(* PLC project FBDexample, Halmstad University FBDexample SNAPSHOT-1.0 *)
(* stored: creationDateTime 2017-08-16T13:43:29, modificationDateTime 2017-08-16T14:46:26 *)

FUNCTION_BLOCK functionBlock0
  VAR
    DBC_PV_CoStep : INT;
    P_Fan1Lo_1 : INT := 3;
    P_Fan1Lo_2 : INT := 7;
    P_Fan1Hi_1 : INT := 8;
    P_Fan2Lo_1 : INT := 4;
    P_Fan2Lo_2 : INT := 6;
    P_Fan2Hi_1 : INT := 7;
    P_Fan2Hi_2 : INT := 8;
    P_Fan3Lo_1 : INT := 5;
    P_Fan3Hi_1 : INT := 6;
    P_Fan3Hi_2 : INT := 8;
    DBC_PV_C_Fan1Lo : BOOL;
    DBC_PV_C_Fan1Hi : BOOL;
    DBC_PV_C_Fan2Lo : BOOL;
    DBC_PV_C_Fan2Hi : BOOL;
    DBC_PV_C_Fan3Lo : BOOL;
    DBC_PV_C_Fan3Hi : BOOL;
  END_VAR

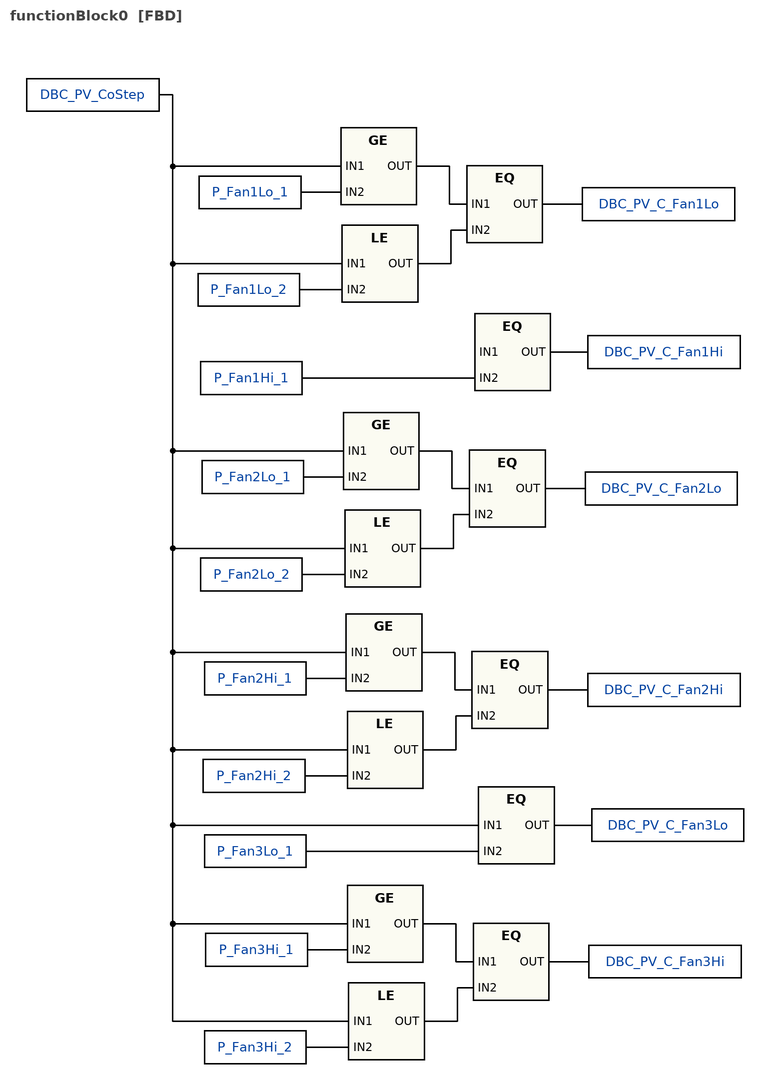
(* FBD diagram, written out as Structured Text *)
DBC_PV_C_Fan1Lo := DBC_PV_CoStep >= P_Fan1Lo_1 = DBC_PV_CoStep <= P_Fan1Lo_2;
DBC_PV_C_Fan1Hi := EQ(IN2 := P_Fan1Hi_1);
DBC_PV_C_Fan2Lo := DBC_PV_CoStep >= P_Fan2Lo_1 = DBC_PV_CoStep <= P_Fan2Lo_2;
DBC_PV_C_Fan2Hi := DBC_PV_CoStep >= P_Fan2Hi_1 = DBC_PV_CoStep <= P_Fan2Hi_2;
DBC_PV_C_Fan3Lo := DBC_PV_CoStep = P_Fan3Lo_1;
DBC_PV_C_Fan3Hi := DBC_PV_CoStep >= P_Fan3Hi_1 = DBC_PV_CoStep <= P_Fan3Hi_2;
END_FUNCTION_BLOCK

FUNCTION_BLOCK functionBlock1
  VAR
    MPW_AV_S_AcmInhSta_Ewa : BOOL;
    MPW_AV_S_AcmInOpr : BOOL;
    MPW_AV_S_AcmInhSta_Ewb : BOOL;
    MPW_AV_S_AcmInOprRm : BOOL;
    Pt_Sep_CtCl : TIME;
    MPV_AV_C_SepCtCl : BOOL;
    TON0 : TON;
  END_VAR
  VAR  (* added by the conversion: wires and edge detectors of the diagram *)
    _NOT6_OUT : BOOL;
  END_VAR

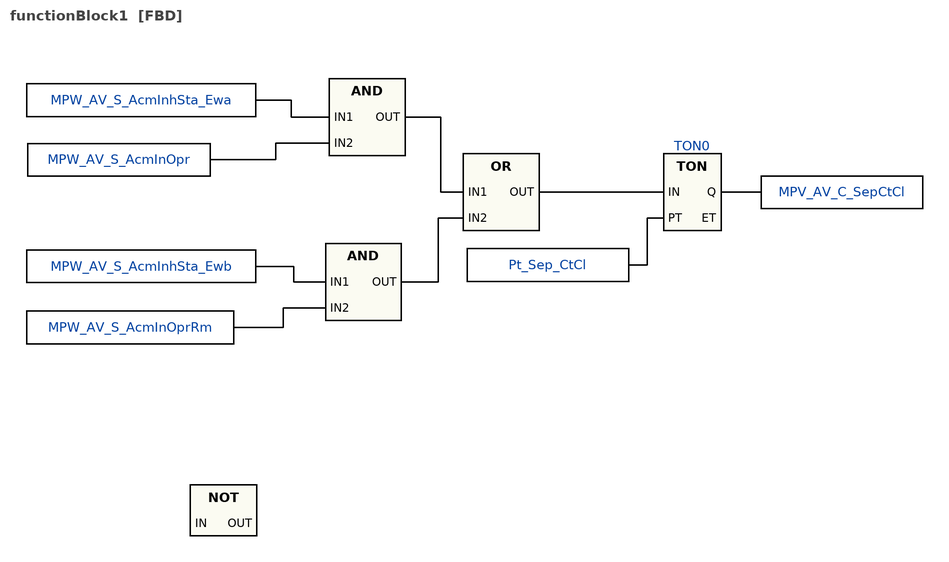
(* FBD diagram, written out as Structured Text *)
TON0(IN := MPW_AV_S_AcmInhSta_Ewa AND MPW_AV_S_AcmInOpr OR MPW_AV_S_AcmInhSta_Ewb AND MPW_AV_S_AcmInOprRm, PT := Pt_Sep_CtCl);
MPV_AV_C_SepCtCl := TON0.Q;
_NOT6_OUT := NOT();
END_FUNCTION_BLOCK
